TYPE F64 : LREAL; END_TYPE

(* stored: Version 1.1.0.1
   DUT F64: Id {3372bce3-0f1d-039e-36aa-16562ff92acf} *)
